FUNCTION_BLOCK FB_LinearActuator_Pneumatic EXTENDS FB_BaseDevice IMPLEMENTS I_Device

VAR
	// Instantiation config variables
	nStroke: INT;
	nAccelMax: INT;			// mm/s2
	nVelocityMax: INT; 		// mm/s
	tExtend: TIME;			// Target time for extend action
	tRetract: TIME;			// Target timef ro retract action
	
	//Output variables
	bOutput_Extend AT %Q*: BOOL;
	bOutput_Retract AT %Q*: BOOL;

	//eSMState:			eMoveState;
	eSMState: (WAIT, EXTEND, RETRACT, STOP, ERROR, RESET) := WAIT;

	tgExecute: 				R_TRIG;
	tTimeout:				TIME := T#3S;
	fbTON_Timeout: TON := 	(PT := tTimeout, IN := FALSE);
END_VAR


VAR_INPUT
	bExecute: BOOL := FALSE;
	eMoveType: E_LinActuatorMoveType;
	fbSwitchExtend:  FB_AutoSwitch;
	fbSwitchRetract: FB_AutoSwitch;
END_VAR

VAR_OUTPUT
	nErrorID: INT;
	bDone: BOOL := FALSE;
END_VAR

tgExecute(CLK := bExecute);
fbTON_Timeout(PT := tTimeout);

IF eStateTarget <> eState AND (bEnable OR (eMode = E_DeviceMode.MANUAL)) THEN
	
	CASE eStateTarget OF 
		E_DeviceState.EXTENDED:
			eMoveType := E_LinActuatorMoveType.EXTEND;
		E_DeviceState.RETRACTED:
			eMoveType := E_LinActuatorMoveType.RETRACT;
		E_DeviceState.IDLE:
			eMoveType := E_LinActuatorMoveType.STOP;
	END_CASE
	bExecute := TRUE;
END_IF


(* move axis using a state machine *)
CASE eSMState OF

	WAIT :	
		// Wait for a command
		IF tgExecute.Q THEN
			CASE eMoveType OF
					E_LinActuatorMoveType.EXTEND:
						eSMState := EXTEND;
					E_LinActuatorMoveType.RETRACT:
						eSMState := RETRACT;
					E_LinActuatorMoveType.STOP:
						eSMState := STOP;
			END_CASE

		END_IF

	EXTEND :
		bOutput_Extend := TRUE;
		bOutput_Retract := FALSE;
		eState := E_DeviceState.EXTENDING;							

		IF fbSwitchExtend.getState() = E_DeviceState.ON THEN
			eState := E_DeviceState.EXTENDED;
			eSMState := WAIT;
			bExecute := FALSE;
		ELSIF fbTON_Timeout.Q THEN
			eSMState := ERROR;
		END_IF

	RETRACT :			
		bOutput_Extend := FALSE;
		bOutput_Retract := TRUE;
		eState := E_DeviceState.RETRACTING;							

		IF fbSwitchRetract.getState() = E_DeviceState.ON THEN
			eState := E_DeviceState.RETRACTED;
			eSMState := WAIT;
			bExecute := FALSE;
		ELSIF fbTON_Timeout.Q THEN
			eSMState := ERROR;
		END_IF
		
	STOP :
		bOutput_Extend := FALSE;
		bOutput_Retract := FALSE;
		eState := E_DeviceState.IDLE;
		bExecute := FALSE;

	ERROR :
		eState := E_DeviceState.FAULTED;
	
END_CASE

METHOD FB_init : BOOL
VAR_INPUT
	bInitRetains : BOOL; // if TRUE, the retain variables are initialized (warm start / cold start)
	bInCopyCode : BOOL;  // if TRUE, the instance afterwards gets moved into the copy code (online change)
	
	Stroke: INT;
	TimeExtend: TIME;
	TimeRetract: TIME;
	
END_VAR
nStroke := Stroke;
tExtend := TimeExtend;
tRetract := TimeRetract;
END_METHOD

END_FUNCTION_BLOCK

(* stored: Version 1.1.0.1, ProductVersion 3.1.4024.12
   POU FB_LinearActuator_Pneumatic: Id {dd7298cc-e501-4f54-b196-3765549d666c}, SpecialFunc None
   Method FB_init: Id {7b20836a-22cf-4c5f-9860-2c3af3af6db5} *)
